// LS Electric XG5000 project: PLC 시험1
// PLC LSPLC
// module base 0 slot 0: 입출력 모듈:XBC-DR14E (DC 24V 입력 8점, 릴레이 출력 6점)

PROGRAM NewProgram (task: 스캔 프로그램)

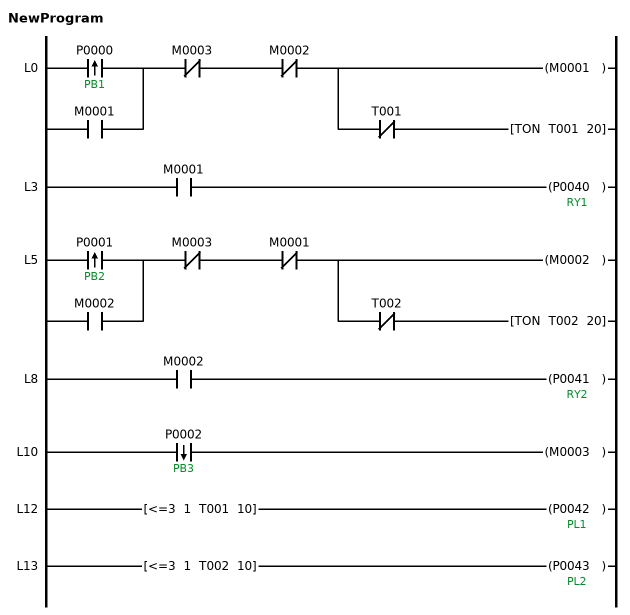
; L0
LOADP     P0000	// PB1
OR        M0001
AND NOT   M0003
AND NOT   M0002
OUT       M0001
AND NOT   T001
TON       T001 20
; L3
LOAD      M0001
OUT       P0040	// RY1
; L5
LOADP     P0001	// PB2
OR        M0002
AND NOT   M0003
AND NOT   M0001
OUT       M0002
AND NOT   T002
TON       T002 20
; L8
LOAD      M0002
OUT       P0041	// RY2
; L10
LOADN     P0002	// PB3
OUT       M0003
; L12
LOAD<=3   1 T001 10
OUT       P0042	// PL1
; L13
LOAD<=3   1 T002 10
OUT       P0043	// PL2